FUNCTION_BLOCK FB_Matrix EXTENDS FB_Device
VAR_INPUT
	st_path : ST_Path;//INT struct to contain int value of path enums
	bSetCurrentPath:BOOL;//Bool to actuate the selected path 
	bPathingOn:BOOL;//BOOL to enable the path selection mode 
	nRowSize:INT;//Matrix row size 
	nColSize:INT;//Matrix Column size
END_VAR
VAR
	aValves:ARRAY [1..4,1..3] OF FB_Solenoid;//Instantiating Solenoid valves, max array size, can contain smaller arrays
	iRows:INT;//Row variable for FOR loops to use
	iColumns:INT;//Col variable for FOR loops to use
	bOverallEnable:BOOL;//Internal variable used to assign device state to all instantiated solenoid valves
END_VAR
VAR_IN_OUT
	aConfig:ARRAY[1..4,1..3] OF ST_SolenoidConfig;//Matrix config
END_VAR
VAR_OUTPUT
	aValveStates : ARRAY [1..4,1..3] OF E_SolenoidState;//State of valves
	aValveCommands:ARRAY [1..4,1..3] OF BOOL;
END_VAR

M_EnableResetLogic();
M_CyclicLogic();
IF bPathingOn THEN
	M_DispensePathing();
ELSE
	M_ManualControl();
END_IF

METHOD M_CyclicLogic : HRESULT
//Call FB_Device M_Cyclic Logic
hr:=SUPER^.M_CyclicLogic();
 IF bDeviceEnable THEN
   FOR iRows := 1 TO nRowSize DO
       FOR iColumns := 1 TO nColSize DO
           aValves[iRows, iColumns](bDeviceEnable:=bOverallEnable,
		   bNormallyOpen:=aConfig[iRows,iColumns].NormallyOpen,
           bCmdOpen:=aConfig[iRows,iColumns].bOpen,bCoilEnergiseState=>aValveCommands[iRows,iColumns]);
       END_FOR
   END_FOR
   
 ELSE
	 FOR iRows := 1 TO nRowSize DO
       FOR iColumns := 1 TO nColSize DO
           aValves[iRows, iColumns](bDeviceEnable:=bOverallEnable);
       END_FOR
     END_FOR
 END_IF
 
FOR iRows := 1 TO nRowSize DO
   FOR iColumns := 1 TO nColSize DO
       aValveStates[iRows, iColumns]:=aValves[iRows, iColumns].eSolenoidState;
   END_FOR
END_FOR
END_METHOD

METHOD M_DispensePathing : BOOL
VAR
	nRowToOpen: INT :=(st_path.startPath);
	nColToOpen: INT :=(st_path.endPath);
END_VAR
IF bDeviceEnable THEN
	IF bSetCurrentPath THEN
       aConfig[nRowToOpen,nColToOpen].bOpen:=TRUE;
    END_IF
END_IF
END_METHOD

METHOD M_EnableResetLogic : BOOL
//Set up variables and logic to reset and enable valve FB's created by FB_Matrix
bOverallEnable:=bDeviceEnable;
IF bDeviceReset THEN
    FOR iRows := 1 TO nRowSize DO
       FOR iColumns := 1 TO nColSize DO
           aValves[iRows, iColumns](bDeviceReset:=fbTrig.Q);
		   aConfig[iRows,iColumns].bOpen:=FALSE;
		   GVL_HMI.aDispManualValveSelection[iRows,iColumns]:=FALSE;
		   GVL_HMI.aInletManualValveSelection[iRows,iColumns]:=FALSE;
		   GVL_HMI.aFillManualValveSelection[iRows,iColumns]:=FALSE;
       END_FOR
    END_FOR
END_IF
END_METHOD

METHOD M_ManualControl
IF NOT bPathingOn AND bDeviceEnable THEN
   FOR iRows := 1 TO 4 DO
       FOR iColumns := 1 TO 3 DO
           aValves[iRows, iColumns](bCmdOpen:=aConfig[iRows,iColumns].bOpen);
       END_FOR
   END_FOR
END_IF
END_METHOD

END_FUNCTION_BLOCK

(* stored: Version 1.1.0.1
   POU FB_Matrix: Id {2c7f537e-a85d-49b4-9066-1d7397aeaf2d}, SpecialFunc None
   Method M_CyclicLogic: Id {f1b117f3-667e-4a24-a226-6ce2e5fb34e4}
   Method M_DispensePathing: Id {1de2314d-8795-4c7a-99e8-ef133b9b0aae}
   Method M_EnableResetLogic: Id {7d457710-3a0c-4071-bb2d-81ff18c2698c}
   Method M_ManualControl: Id {0be0b670-86a1-4a84-85ca-54c8277a37d4} *)
